INTERFACE I_PtDateTime

END_INTERFACE

(* stored: Version 1.1.0.1, ProductVersion 3.1.4024.12
   Itf I_PtDateTime: Id {11593b05-65e3-4a1a-b9a6-9e055a74fa99} *)
